// TIA Portal V17 export
// export: Created 2025-03-10T12:16:28.7614243Z, ExportSetting WithDefaults, DisplayName Totally Integrated Automation Portal, DisplayVersion V17 Update 8, DisplayName TIA Portal Openness, DisplayVersion V17 Update 8, DisplayName TIA Portal Version Control Interface, DisplayVersion V17, DisplayName SINAMICS Startdrive Advanced, DisplayVersion V17 SP2, DisplayName SINAMICS Startdrive G110M, G120, G120C, G120D, G120P, G115D, DisplayVersion V17 SP2, DisplayName SINAMICS Startdrive G130, G150, S120, S150, SINAMICS MV, S210, DisplayVersion V17 SP2, DisplayName STEP 7 Professional, DisplayVersion V17 Update 8, DisplayName SINUMERIK ONE STEP 7 Toolbox, DisplayVersion V17 Update 12, DisplayName SINUMERIK 840D sl STEP 7 Toolbox, DisplayVersion V17 Update 12, DisplayName STEP 7 Safety, DisplayVersion V17 Update 6, DisplayName WinCC Advanced, DisplayVersion V17 Update 8
FUNCTION "FC1400_SERVICES_GENERAL" : Void   // FC1400, LAD
{ S7_Optimized_Access := 'FALSE' }
AUTHOR : ETXETAR
VERSION : 1.0
// stored: AutoNumber false, IsIECCheckEnabled false, SetENOAutomatically false, UDAEnableTagReadback false
BEGIN

REGION Network 1: CALL FC1401_UTILITY_SKIDS
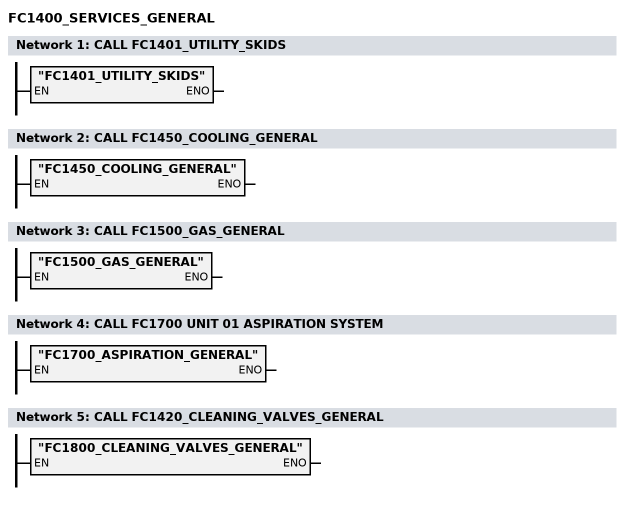
   RUNG wire#powerrail
      "FC1401_UTILITY_SKIDS"()
   END_RUNG
   // the same network as SCL:
   "FC1401_UTILITY_SKIDS"();
END_REGION

REGION Network 2: CALL FC1450_COOLING_GENERAL
   RUNG wire#powerrail
      "FC1450_COOLING_GENERAL"()
   END_RUNG
   // the same network as SCL:
   "FC1450_COOLING_GENERAL"();
END_REGION

REGION Network 3: CALL FC1500_GAS_GENERAL
   RUNG wire#powerrail
      "FC1500_GAS_GENERAL"()
   END_RUNG
   // the same network as SCL:
   "FC1500_GAS_GENERAL"();
END_REGION

REGION Network 4: CALL FC1700 UNIT 01 ASPIRATION SYSTEM
   RUNG wire#powerrail
      "FC1700_ASPIRATION_GENERAL"()
   END_RUNG
   // the same network as SCL:
   "FC1700_ASPIRATION_GENERAL"();
END_REGION

REGION Network 5: CALL FC1420_CLEANING_VALVES_GENERAL
   RUNG wire#powerrail
      "FC1800_CLEANING_VALVES_GENERAL"()
   END_RUNG
   // the same network as SCL:
   "FC1800_CLEANING_VALVES_GENERAL"();
END_REGION
END_FUNCTION
